SUBAPPLICATION DO_TOGGLE_RPC_QXA_OPC (* Digitaler Freigabe-Ausgang als Klick-Toggle (AX_T_FF_INIT, Default AN): CREATE_METHOD-Server nimmt einen argumentlosen RPC-Trigger von mehreren gleichberechtigten Aufrufern entgegen (z.B. STG1-SoftKey-Relay UND OPC-Dashboard), alle takten denselben CLK - KEIN OR nach dem Flipflop, AX_T_FF_INIT.Q ist alleinige Source of Truth fuer den physischen Ausgang UND den remote publizierten Zustand. Generisch fuer jeden Not-Bedienung-/Strassenmodus-artigen Digital-Toggle-Ausgang mit Mehrfach-Bedienung. *)
  (* Standard: 61499-2 *)
  (* Version 1.0, 2026-09-08, Franz Höpfinger, Meisterschulen am Ostbahnhof, Ausgelagert aus Heben_Senken_TO_QDA_PWM_OPC (Freigabe-DO-Teilnetz) zur Wiederverwendung fuer weitere Digital-Toggle-Ausgaenge. *)
  PACKAGE MyLib::sys;
  IMPORT logiBUS::io::DQ::logiBUS_DO;
  IMPORT logiBUS::io::DQ::logiBUS_DO_S;
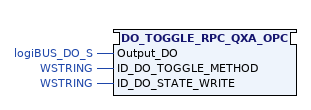
  VAR_INPUT
    Output_DO : logiBUS::io::DQ::logiBUS_DO_S := logiBUS_DO::Invalid; (* Physischer Freigabe-Ausgang: Klick-Toggle, Default AN *)
    ID_DO_TOGGLE_METHOD : WSTRING; (* Lokale Methodenadresse (ACTION=CREATE_METHOD) fuer den argumentlosen Freigabe-Toggle-Trigger - wird von mehreren Aufrufern gemeinsam genutzt, alle takten denselben Flipflop *)
    ID_DO_STATE_WRITE : WSTRING; (* Lokale Publish-Adresse (ACTION=WRITE) fuer den tatsaechlichen Freigabe-Zustand (AX_T_FF_INIT.Q) - wird remote abonniert *)
  END_VAR
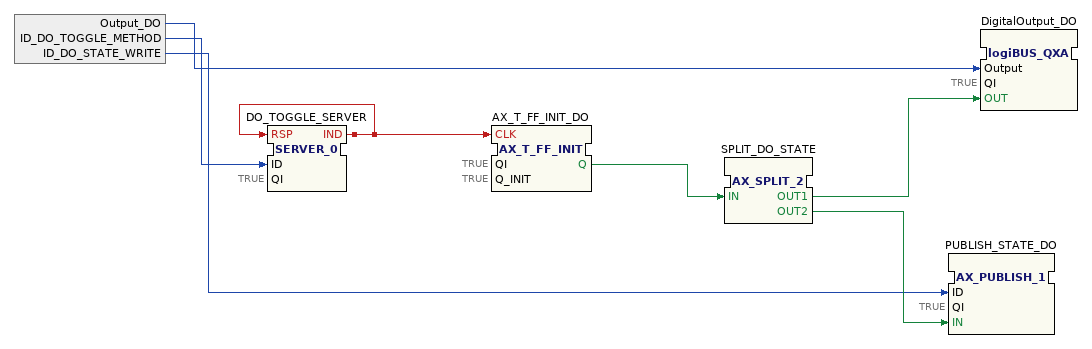
  (* AX_T_FF_INIT.Q ist die EINZIGE Source of Truth fuer DigitalOutput_DO - KEIN AX_OR_2 nach dem Flipflop (anders als TOGGLE_RPC_MERGE_QXA_OPC/Blitzer). Der Methodenaufruf (ID_DO_TOGGLE_METHOD) ist der einzige Eingang und wird von mehreren Aufrufern gemeinsam genutzt - alle takten denselben CLK, kein Merge auf Datenebene noetig. *)
  (* RSP MUSS auf IND zurueckverdrahtet werden (argumentloser Trigger, keine Verarbeitung noetig - wie FORTEs eigener systemtests/clientFailAction.fboot: IND->RSP direkt). Ohne RSP blockiert FORTEs onServerMethodCall den OPC-UA-Server-Thread bis zu 4s (scmMethodCallTimeoutInNanoSeconds) und haelt dabei open62541s globalen serviceMutex - der von JEDEM AX_PUBLISH_1 auf einem anderen FORTE-Thread ebenfalls gebraucht wird. Folge: physischer Ausgang reagiert sofort (kein Lock noetig), aber JEDE OPC-UA-Statusmeldung (nicht nur diese hier) haengt bis zu 4s fest. Siehe Ventilsteuerung/OPC_UA_VERNETZUNG.md Punkt 12. *)
  FBS
    DO_TOGGLE_SERVER : iec61499::net::SERVER_0(QI := TRUE);
    AX_T_FF_INIT_DO : adapter::events::unidirectional::AX_T_FF_INIT(QI := TRUE, Q_INIT := TRUE);
    SPLIT_DO_STATE : adapter::events::unidirectional::AX_SPLIT_2;
    PUBLISH_STATE_DO : adapter::net::AX_PUBLISH_1(QI := TRUE);
    DigitalOutput_DO : logiBUS::io::DQ::logiBUS_QXA(QI := TRUE);
  END_FBS
  EVENT_CONNECTIONS
    DO_TOGGLE_SERVER.IND TO AX_T_FF_INIT_DO.CLK;
    DO_TOGGLE_SERVER.IND TO DO_TOGGLE_SERVER.RSP;
  END_CONNECTIONS
  DATA_CONNECTIONS
    Output_DO TO DigitalOutput_DO.Output;
    ID_DO_TOGGLE_METHOD TO DO_TOGGLE_SERVER.ID;
    ID_DO_STATE_WRITE TO PUBLISH_STATE_DO.ID;
  END_CONNECTIONS
  ADAPTER_CONNECTIONS
    AX_T_FF_INIT_DO.Q TO SPLIT_DO_STATE.IN;
    SPLIT_DO_STATE.OUT1 TO DigitalOutput_DO.OUT;
    SPLIT_DO_STATE.OUT2 TO PUBLISH_STATE_DO.IN;
  END_CONNECTIONS
END_SUBAPPLICATION
